(* Logix 5000 project; controller Safety vendor 1 type 14 code 86 rev 19.11; software revision 19.01; part 2 of 17 *)
(* tags used below, declared in another part *)
   A1_IO : UDT_CardSts[32];   // A1 Point I/O
   A1_IOSts_Flt : BOOL;   // A1 Point IO Module Fault ( 1= Faulted)
   C1_IO : UDT_CardSts[32];   // C1 Point I/O
   C1_IOSts_Flt : BOOL;   // C1 Point IO Module Fault ( 1= Faulted)
   CHPLC_IO : UDT_CardSts[32];   // CHPLC Point I/O
   CHPLC_IOSts_Flt : BOOL;   // CHPLC Point IO Module Fault ( 1= Faulted)
   D1_IO : UDT_CardSts[32];   // D1 Point I/O
   D1_IOSts_Flt : BOOL;   // D1 Point IO Module Fault ( 1= Faulted)
   DPD_IO : UDT_CardSts[32];   // DPD Point I/O
   DPD_IOSts_Flt : BOOL;   // DPD Point IO Module Fault ( 1= Faulted)
   E1_IO : UDT_CardSts[32];   // E1 Point I/O
   E1_IOSts_Flt : BOOL;   // E1 Point IO Module Fault ( 1= Faulted)
   F1_IO : UDT_CardSts[32];   // F1 Point I/O
   F1_IOSts_Flt : BOOL;   // F1 Point IO Module Fault ( 1= Faulted)
   Flt_Modules : DINT[5];   // Point IO Module Fault Word
   G1_IO : UDT_CardSts[32];   // G1 Point I/O
   G1_IOSts_Flt : BOOL;   // G1 Point IO Module Fault ( 1= Faulted)
   H1_IO : UDT_CardSts[32];   // H1 Point I/O
   H1_IOSts_Flt : BOOL;   // H1 Point IO Module Fault ( 1= Faulted)
   Line_TotalMode : BOOL;   // Line TOTAL Mode ( 1= Total Mode) (0 = Coil to Coil)
   LineSts : UDT_SysStatus;
   Local_ModFlts : DINT;   // Local Card Fault Status
   Local_Networks_OK : BOOL;   // Local Network CARDS OK ( 1= OK)
   Local_Slot : UDT_CardSts[17];   // Safety Processor
   MCC1_IO : UDT_CardSts[32];   // MCC1 Point I/O
   MCC1_IOSts_Flt : BOOL;   // MCC1 Point IO Module Fault ( 1= Faulted)
   MCC3_IO : UDT_CardSts[32];   // MCC3 Point I/O
   MCC4_IO : UDT_CardSts[32];   // MCC4 Point I/O
   OS11_IO : UDT_CardSts[32];   // OS11 Point I/O
   OS13_IO : UDT_CardSts[32];   // OS13 Point I/O
   OS14_IO : UDT_CardSts[32];   // OS14 Point I/O
   OS15_IO : UDT_CardSts[32];   // OS15 Point I/O
   OS16_IO : UDT_CardSts[32];   // OS16 Point I/O
   OS1_IO : UDT_CardSts[32];   // OS1 Point I/O
   OS2_IO : UDT_CardSts[32];   // OS2 Point I/O
   OS3_IO : UDT_CardSts[32];   // OS3 Point I/O
   OS4N_IO : UDT_CardSts[32];   // OS4N Point I/O
   OS4S_IO : UDT_CardSts[32];   // OS4S Point I/O
   OS5_IO : UDT_CardSts[32];   // OS5 Point I/O
   OS6_IO : UDT_CardSts[32];   // OS6 Point I/O
   OS8_IO : UDT_CardSts[32];   // OS8 Point I/O
   OS9_IO : UDT_CardSts[32];   // OS9 Point I/O
   Peer_Networks_OK : BOOL;   // Peer Network CARDS OK ( 1= OK)
   Rem_ModFlts : DINT;   // Remote IO Comm Faults
   SDPLC_IO : UDT_CardSts[32];   // SDPLC Point I/O
   SftyMap_Mach : DINT[5];   // SAFETY MAPPED From Machine Processor
   Sy_ClrFlt : BOOL;   // System Clear Fault

   UNW_SafeOffFltRst : BOOL;   // Unwind Safe-Off Fault Reset ( 1= Reset Cmd )
   UnwHoldDwn_FVR_En : BOOL := 1;   // Unwind Hold Down Roll FVR Enable ( 1= Enable )
   UnwHoldDwn_FVR_FltRst : BOOL;   // Unwind Hold Down Roll Fault Reset ( 1= Reset Cmd )
   UnwHoldDwn_FVR_FwdCmd : BOOL;   // Unwind Hold Down Roll Forward Command ( 1= Run Fwd )
   UnwHoldDwn_FVR_RevCmd : BOOL;   // Unwind Hold Down Roll Reverse Command ( 1= Run Rev)
   UWCC_Rst_PB : ALIAS FOR SftyMap_Mach[0].10;   // Unwind Coil Car Safety Reset PB
   VS2_IO : UDT_CardSts[32] := ([0].EntrySts := 16897, [0].Running := 1);   // VS2 Point I/O
        [4]   // 1734-IE2C/C
   VS2_IOSts_Flt : BOOL;   // VS2 Point IO Module Fault ( 1= Faulted)
   VS2_S10_ModFlt : ALIAS FOR Flt_Modules[0].21;   // VS2 Point I/O Slot10 Module Fault (1 = Fault)
   VS2_SolPwrEn : BOOL := 1;   // VS2 Solenoid Safe-Off Enable ( 1= Enable )
   WTPR_DrvsOff : BOOL;   // Wash Tank Pinch Rolls (1-4) Drives OFF ( 1= OFF)
   WTPR_SafeTrqEn : BOOL := 1;   // Wash Tank Pinch Rolls (1-4) Safe-Trq Off Enable ( 1= Enable )
   x172CR460 : ALIAS FOR SDPLC:1:I.Pt00Data;   // Shear Die Drive Main Contactor Safety Relay Input
   x172CR510 : ALIAS FOR SDPLC:1:I.Pt01Data;   // Shear Die Drive Enable Safety Relay Input
   x201PB040a : ALIAS FOR OS1:1:I.Pt00Data;   // Line Emergency Stop PB
   x201PB040b : ALIAS FOR OS1:1:I.Pt01Data;   // Line Emergency Stop PB
   x211PB040a : ALIAS FOR OS2:1:I.Pt00Data;   // Line Emergency Stop PB
   x211PB040b : ALIAS FOR OS2:1:I.Pt01Data;   // Line Emergency Stop PB
   x221PB040a : ALIAS FOR OS3:1:I.Pt00Data;   // Emergency Stop PB
   x221PB040b : ALIAS FOR OS3:1:I.Pt01Data;   // Emergency Stop PB
   x231PB040a : ALIAS FOR OS4N:1:I.Pt00Data;   // Emergency Stop PB
   x231PB040b : ALIAS FOR OS4N:1:I.Pt01Data;   // Emergency Stop PB
   x241PB040a : ALIAS FOR OS4S:1:I.Pt00Data;   // Emergency Stop PBMc_A_Run1_A
   x241PB040b : ALIAS FOR OS4S:1:I.Pt01Data;   // Emergency Stop PBMc_A_Run1_A
   x251PB040a : ALIAS FOR OS5:1:I.Pt00Data;   // Emergency Stop PB
   x251PB040b : ALIAS FOR OS5:1:I.Pt01Data;   // Emergency Stop PB
   x261PB040a : ALIAS FOR OS6:1:I.Pt00Data;   // Emergency Stop PB
   x261PB040b : ALIAS FOR OS6:1:I.Pt01Data;   // Emergency Stop PB
   x271PB040a : ALIAS FOR OS8:1:I.Pt00Data;   // Emergency Stop PB
   x271PB040b : ALIAS FOR OS8:1:I.Pt01Data;   // Emergency Stop PB
   x281PB040a : ALIAS FOR OS9:1:I.Pt00Data;   // Emergency Stop PB
   x281PB040b : ALIAS FOR OS9:1:I.Pt01Data;   // Emergency Stop PB
   x291PB040a : ALIAS FOR OS11:1:I.Pt00Data;   // Emergency Stop PB
   x291PB040b : ALIAS FOR OS11:1:I.Pt01Data;   // Emergency Stop PB
   x301PB040a : ALIAS FOR OS13:1:I.Pt00Data;   // Emergency Stop PB
   x301PB040b : ALIAS FOR OS13:1:I.Pt01Data;   // Emergency Stop PB
   x301PBL500 : BOOL;   // Tandem Jog PBL
   x301SS540a : BOOL;   // Sheeter Pinch Roll Jog Forward SS
   x301SS540b : BOOL;   // Sheeter Pinch Roll Jog Reverse SS
   x311PB040a : ALIAS FOR OS14:1:I.Pt00Data;   // Emergency Stop PB OS14
   x311PB040b : ALIAS FOR OS14:1:I.Pt01Data;   // Emergency Stop PB OS14
   x311PB130a : ALIAS FOR OS14:1:I.Pt02Data;   // Shear Emergency Stop PB Os14
   x311PB130b : ALIAS FOR OS14:1:I.Pt03Data;   // Shear Emergency Stop PB Os14
   x312PB700 : BOOL;   // Product Conveyor Jog Forward PB
   x312PB740 : BOOL;   // Product Conveyor Jog Reverse PB
   x312SS460a : BOOL;   // Scrap Conveyor Jog Forward SS
   x312SS460b : BOOL;   // Scrap Conveyor Jog Reverse SS
   x313PBL080 : BOOL;   // Tandem Jog PBL
   x313SS460a : BOOL;   // Shear Conveyor Jog Forward SS
   x313SS460b : BOOL;   // Shear Conveyor Jog Reverse SS
   x314SS040a : BOOL;   // Shear Pinch Roll Jog Forward SS
   x314SS040b : BOOL;   // Shear Pinch Roll Jog Reverse SS
   x315SS040a : BOOL;   // Sheeter Pinch Roll Jog Forward SS
   x315SS040b : BOOL;   // Sheeter Pinch Roll Jog Reverse SS
   x321PB040a : ALIAS FOR OS15:1:I.Pt00Data;   // Emergency Stop PB
   x321PB040b : ALIAS FOR OS15:1:I.Pt01Data;   // Emergency Stop PB
   x331PB040a : ALIAS FOR OS16:1:I.Pt00Data;   // Emergency Stop PB
   x331PB040b : ALIAS FOR OS16:1:I.Pt01Data;   // Emergency Stop PB
   x406LCA047 : ALIAS FOR A1:21:I.Pt00Data;   // North/South Light Curtain Output A
   x406LCB052 : ALIAS FOR A1:21:I.Pt01Data;   // North/South Light Curtain Output B
   x480PB470a : ALIAS FOR DPD:15:I.Pt00Data;   // Emergency Stop Pushbutton
   x480PB470b : ALIAS FOR DPD:15:I.Pt01Data;   // Emergency Stop Pushbutton
   x480PB550a : ALIAS FOR DPD:15:I.Pt02Data;   // Emergency Stop Pushbutton (In Pit)
   x480PB550b : ALIAS FOR DPD:15:I.Pt03Data;   // Emergency Stop Pushbutton (In Pit)
   x519LS470 : ALIAS FOR G1:12:I.Pt00Data;   // Tripwire Emergency Stop Limit Switch
   x533PB470a : ALIAS FOR H1:6:I.Pt00Data;   // Sheeter Emergency Stop Pushbutton
   x533PB470b : ALIAS FOR H1:6:I.Pt01Data;   // Sheeter Emergency Stop Pushbutton
   x613CR460 : ALIAS FOR CHPLC:1:I.Pt00Data;   // Unwind Operator Side Main Contactor Safety Relay
   x613CR510 : ALIAS FOR CHPLC:1:I.Pt01Data;   // Unwind Operator Side Drive Enable Safety Relay
   x613CR550 : ALIAS FOR CHPLC:1:I.Pt02Data;   // Unwind Drive Side Main Contactor Safety Relay
   x613CR590 : ALIAS FOR CHPLC:1:I.Pt03Data;   // Unwind Drive Side Drive Enable Safety Relay
   x613CR630 : ALIAS FOR CHPLC:1:I.Pt04Data;   // #1 Entry Bridle Roll 2 Main Contactor Safety Relay
   x613CR670 : ALIAS FOR CHPLC:1:I.Pt05Data;   // #1 Entry Bridle Roll 2 Drive Enable Safety Relay
   x613CR710 : ALIAS FOR CHPLC:1:I.Pt06Data;   // #2 Entry Bridle Roll 3 Main Contactor Safety Relay
   x613CR750 : ALIAS FOR CHPLC:1:I.Pt07Data;   // #2 Entry Bridle Roll 3 Drive Enable Safety Relay
   x614CR040 : ALIAS FOR CHPLC:2:I.Pt00Data;   // #1 Exit Bridle Roll 6 Main Contactor Safety Relay
   x614CR090 : ALIAS FOR CHPLC:2:I.Pt01Data;   // #1 Exit Bridle Roll 6 Drive Enable Safety Relay
   x614CR130 : ALIAS FOR CHPLC:2:I.Pt02Data;   // #2 Exit Bridle Roll 7 Main Contactor Safety Relay
   x614CR170 : ALIAS FOR CHPLC:2:I.Pt03Data;   // #2 Exit Bridle Roll 7 Drive Enable Safety Relay
   x614CR210 : ALIAS FOR CHPLC:2:I.Pt04Data;   // Rewind Main Contactor Safety Relay
   x614CR250 : ALIAS FOR CHPLC:2:I.Pt05Data;   // Rewind Drive Enable Safety Relay
   x702MTR191FF : ALIAS FOR MCC1:1:I.Pt00Data;   // Rewind Pinch Roll Fwd Fdbk
   x702MTR191RF : ALIAS FOR MCC1:1:I.Pt01Data;   // Rewind Pinch Roll Rev Fdbk
   x708MTR080FF : ALIAS FOR MCC1:1:I.Pt04Data;   // Flattener Drive Motor Fwd Fdbk
   x708MTR080RF : ALIAS FOR MCC1:1:I.Pt05Data;   // Flattener Drive Motor Rev Fdbk
   x708MTR250FF : ALIAS FOR MCC1:1:I.Pt06Data;   // Unwind Holddown Roll Drive Motor Fwd Fdbk
   x708MTR250RF : ALIAS FOR MCC1:1:I.Pt07Data;   // Unwind Holddown Roll Drive Motor Rev Fdbk
   x753MTR190FF : ALIAS FOR MCC3:1:I.Pt00Data;   // Trimmer Pinch Roll Fwd Fdbk
   x753MTR190RF : ALIAS FOR MCC3:1:I.Pt01Data;   // Trimmer Pinch Roll Rev Fdbk
   x759MTR080SE : ALIAS FOR MCC3:4:O.Pt02Data;   // Scrap Choppers Width Adjust Safety Enable
   x759MTR080SP : ALIAS FOR MCC3:4:O.Pt01Data;   // Scrap Choppers Width Adjust Safety Power
   x761MTR081RF : ALIAS FOR MCC3:1:I.Pt02Data;   // Trimmer Scrap Conveyor RunFdbk
   x775MTR280RF : BOOL := 1;   // (From Shear DIe) Shear Pinch Roll Lube Run Fdbk
   x778MTR080RF : ALIAS FOR MCC4:1:I.Pt00Data;   // Shear Crank Motor Run Fdbk
   x781MTR080RF : BOOL := 1;   // (From Shear DIe) Sheeter Pinch Roll Lube Run Fdbk
   x781MTR190RF : BOOL := 1;   // (From Shear DIe) Sheeter Hyd Pump Run Fdbk
   x802MTR080FF : ALIAS FOR MCC5:1:I.Pt00Data;   // Stacker Side Guide Lift Fwd Fdbk/Up
   x802MTR080RF : ALIAS FOR MCC5:1:I.Pt01Data;   // Stacker Side Guide Lift Rev Fdbk/Down
   x802MTR230FF : ALIAS FOR MCC5:1:I.Pt02Data;   // Scrap Horizontal Conveyor Run Fwd Fdbk
   x802MTR230RF : ALIAS FOR MCC5:1:I.Pt03Data;   // Scrap Horizontal Conveyor Run Rev Fdbk
   x802MTR231FF : ALIAS FOR MCC5:1:I.Pt04Data;   // Stacker Chain Fwd Fdbk
   x802MTR231RF : ALIAS FOR MCC5:1:I.Pt05Data;   // Stacker Chain Rev Fdbk
   x813MTR080RF : BOOL := 1;   // (From Shear DIe) Exit Conveyor Hyd Pump Run Fdbk
   y172CR460 : ALIAS FOR SDPLC:2:O.Pt00Data;   // Shear Die Drive Main Contactor Safety Relay Output
   y172CR510 : ALIAS FOR SDPLC:2:O.Pt01Data;   // Shear Die Drive Enable Safety Relay Output
   y172CR550 : ALIAS FOR SDPLC:2:O.Pt02Data;   // Line Soleniod Safe-Off
   y233CR040 : ALIAS FOR OS4N:5:O.Pt00Data;   // OS4N Solenoid Safe Off
   y243CR040 : ALIAS FOR OS4S:5:O.Pt00Data;   // OS4S Solenoid Safe Off
   y406CR050 : ALIAS FOR A1:20:O.Pt00Data;   // Line Solenoid Safe Off
   y406CR090 : ALIAS FOR A1:20:O.Pt01Data;   // Coil Car Solenoid Safe Off
   y406CR120 : ALIAS FOR A1:20:O.Pt02Data;   // Spare
   y406CR170 : ALIAS FOR A1:20:O.Pt03Data;   // Spare
   y435CR050 : ALIAS FOR C1:12:O.Pt00Data;   // Solenoid Safe Off
   y451CR050 : ALIAS FOR D1:12:O.Pt00Data;   // Soleniod Safe Off
   y464CR050 : ALIAS FOR E1:10:O.Pt00Data;   // Soleniod Safe Off
   y480CR050 : ALIAS FOR DPD:14:O.Pt00Data;   // Solenoid Safe Off
   y495CR050 : ALIAS FOR VS2:10:O.Pt00Data;   // Soleniod Safe Off
   y507CR050 : ALIAS FOR F1:19:O.Pt00Data;   // Line Solenoid Safe Off
   y507CR090 : ALIAS FOR F1:19:O.Pt01Data;   // Rewind Coil Car Solenoid Safe Off
   y519CR050 : ALIAS FOR G1:11:O.Pt00Data;   // Line Solenoid Safe Off
   y533CR050 : ALIAS FOR H1:5:O.Pt00Data;   // Line Solenoid Safe Off
   y613CR460 : ALIAS FOR CHPLC:4:O.Pt00Data;   // Unwind Operator Side Main Contactor Safety Relay
   y613CR510 : ALIAS FOR CHPLC:4:O.Pt01Data;   // Unwind Operator Side Drive Enable Safety Relay
   y613CR550 : ALIAS FOR CHPLC:4:O.Pt02Data;   // Unwind Drive Side Main Contactor Safety Relay
   y613CR590 : ALIAS FOR CHPLC:4:O.Pt03Data;   // Unwind Drive Side Drive Enable Safety Relay
   y613CR630 : ALIAS FOR CHPLC:4:O.Pt04Data;   // #1 Entry Bridle Roll 2 Main Contactor Safety Relay
   y613CR670 : ALIAS FOR CHPLC:4:O.Pt05Data;   // #1 Entry Bridle Roll 2 Drive Enable Safety Relay
   y613CR710 : ALIAS FOR CHPLC:4:O.Pt06Data;   // #2 Entry Bridle Roll 3 Main Contactor Safety Relay
   y613CR750 : ALIAS FOR CHPLC:4:O.Pt07Data;   // #2 Entry Bridle Roll 3 Drive Enable Safety Relay
   y614CR040 : ALIAS FOR CHPLC:5:O.Pt00Data;   // #1 Exit Bridle Roll 6 Main Contactor Safety Relay
   y614CR090 : ALIAS FOR CHPLC:5:O.Pt01Data;   // #1 Exit Bridle Roll 6 Drive Enable Safety Relay
   y614CR130 : ALIAS FOR CHPLC:5:O.Pt02Data;   // #2 Exit Bridle Roll 7 Main Contactor Safety Relay
   y614CR170 : ALIAS FOR CHPLC:5:O.Pt03Data;   // #2 Exit Bridle Roll 7 Drive Enable Safety Relay
   y614CR210 : ALIAS FOR CHPLC:5:O.Pt04Data;   // Rewind Main Contactor Safety Relay
   y614CR250 : ALIAS FOR CHPLC:5:O.Pt05Data;   // Rewind Drive Enable Safety Relay
   y702MTR191FC : ALIAS FOR MCC1:6:O.Pt00Data;   // Rewind Pinch Roll Fwd Cmd
   y702MTR191RC : ALIAS FOR MCC1:6:O.Pt01Data;   // Rewind Pinch Roll Rev Cmd
   y708MTR080FC : ALIAS FOR MCC1:6:O.Pt04Data;   // Flattener Drive Motor Fwd Cmd
   y708MTR080RC : ALIAS FOR MCC1:6:O.Pt05Data;   // Flattener Drive Motor Rev Cmd
   y708MTR250FC : ALIAS FOR MCC1:6:O.Pt06Data;   // Unwind Holddown Roll Drive Motor Fwd Cmd
   y708MTR250RC : ALIAS FOR MCC1:6:O.Pt07Data;   // Unwind Holddown Roll Drive Motor Rev Cmd
   y725MTR080SE : ALIAS FOR MCC2:1:O.Pt01Data;   // Unwind Pinch Roll Safety Enable
   y725MTR080SP : ALIAS FOR MCC2:1:O.Pt00Data;   // Unwind Pinch Roll Safety Power
   y727MTR080SE : ALIAS FOR MCC2:1:O.Pt05Data;   // Paper Winder Safety Enable
   y727MTR080SP : ALIAS FOR MCC2:1:O.Pt04Data;   // Paper Winder Safety Power
   y729MTR080SE : ALIAS FOR MCC2:1:O.Pt03Data;   // Washtank Pinch Roll 4 Safety Enable
   y729MTR080SP : ALIAS FOR MCC2:1:O.Pt02Data;   // Washtank Pinch Roll 4 Safety Power
   y731MTR080SE : ALIAS FOR MCC2:1:O.Pt07Data;   // Washtank Pinch Roll 1 Safety Enable
   y731MTR080SP : ALIAS FOR MCC2:1:O.Pt06Data;   // Washtank Pinch Roll 1 Safety Power
   y733MTR080SE : ALIAS FOR MCC2:2:O.Pt01Data;   // Washtank Pinch Roll 2 Safety Enable
   y733MTR080SP : ALIAS FOR MCC2:2:O.Pt00Data;   // Washtank Pinch Roll 2 Safety Power
   y735MTR080SE : ALIAS FOR MCC2:2:O.Pt03Data;   // Washtank Pinch Roll 3 Safety Enable
   y735MTR080SP : ALIAS FOR MCC2:2:O.Pt02Data;   // Washtank Pinch Roll 3 Safety Power
   y751MTR080SE : ALIAS FOR MCC3:3:O.Pt04Data;   // Trimmer Knives Safety Enable
   y751MTR080SP : ALIAS FOR MCC3:3:O.Pt03Data;   // Trimmer Knives Safety Power
   y753MTR190FC : ALIAS FOR MCC3:3:O.Pt00Data;   // Trimmer Pinch Roll Fwd Cmd
   y753MTR190RC : ALIAS FOR MCC3:3:O.Pt01Data;   // Trimmer Pinch Roll Rev Cmd
   y754MTR080SE : ALIAS FOR MCC3:3:O.Pt06Data;   // Side Guide Width Adjust Safety Enable
   y754MTR080SP : ALIAS FOR MCC3:3:O.Pt05Data;   // Side Guide Width Adjust Safety Power
   y755MTR080SE : ALIAS FOR MCC3:4:O.Pt00Data;   // Trimmer Knives Width Adjust Safety Enable
   y755MTR080SP : ALIAS FOR MCC3:3:O.Pt07Data;   // Trimmer Knives Width Adjust Safety Power
   y761MTR081RC : ALIAS FOR MCC3:3:O.Pt02Data;   // Trimmer Scrap Conveyor RunCmd
   y762MTR080SE : ALIAS FOR MCC3:4:O.Pt04Data;   // Scrap Choppers Safety Enable
   y762MTR080SP : ALIAS FOR MCC3:4:O.Pt03Data;   // Scrap Choppers Safety Power
   y776MTR080SE : ALIAS FOR MCC4:3:O.Pt07Data;   // Shear Metering Backup Roll Safety Enable
   y776MTR080SP : ALIAS FOR MCC4:3:O.Pt06Data;   // Shear Metering Backup Roll Safety Power
   y778MTR080RC : ALIAS FOR MCC4:4:O.Pt00Data;   // Shear Die Crank Run Cmd
   y779MTR080SE : ALIAS FOR MCC4:3:O.Pt01Data;   // Shear Pinch Roll Safety Enable
   y779MTR080SP : ALIAS FOR MCC4:3:O.Pt00Data;   // Shear Pinch Roll Safety Power
   y782MTR080SE : ALIAS FOR MCC4:3:O.Pt03Data;   // Sheeter Pinch Roll Safety Enable
   y782MTR080SP : ALIAS FOR MCC4:3:O.Pt02Data;   // Sheeter Pinch Roll Safety Power
   y785MTR080SE : ALIAS FOR MCC4:3:O.Pt05Data;   // Stacker Blower Safety Enable
   y785MTR080SP : ALIAS FOR MCC4:3:O.Pt04Data;   // Stacker Blower Safety Power
   y800MTR080SE : ALIAS FOR MCC5:3:O.Pt01Data;   // Scrap Incline Conveyor Safety Enable
   y800MTR080SP : ALIAS FOR MCC5:3:O.Pt00Data;   // Scrap Incline Conveyor Safety Power
   y802MTR080FC : ALIAS FOR MCC5:4:O.Pt04Data;   // Stacker Side Guide Lift Fwd Cmd/Up
   y802MTR080RC : ALIAS FOR MCC5:4:O.Pt05Data;   // Stacker Side Guide Lift Rev Cmd/Down
   y802MTR230FC : ALIAS FOR MCC5:4:O.Pt06Data;   // Scrap Horizontal Conveyor Fwd Cmd
   y802MTR230RC : ALIAS FOR MCC5:4:O.Pt07Data;   // Scrap Horizontal Conveyor Rev Cmd
   y802MTR231FC : ALIAS FOR MCC5:5:O.Pt00Data;   // Stacker Chain Fwd Cmd
   y802MTR231RC : ALIAS FOR MCC5:5:O.Pt01Data;   // Stacker Chain Rev Cmd
   y804MTR080SE : ALIAS FOR MCC5:3:O.Pt03Data;   // Stacker Back Stop Safety Enable
   y804MTR080SP : ALIAS FOR MCC5:3:O.Pt02Data;   // Stacker Back Stop Safety Power
   y806MTR080SE : ALIAS FOR MCC5:3:O.Pt05Data;   // Product Conveyor 3 Safety Enable
   y806MTR080SP : ALIAS FOR MCC5:3:O.Pt04Data;   // Product Conveyor 3 Safety Power
   y808MTR080SE : ALIAS FOR MCC5:3:O.Pt07Data;   // Product Conveyor 1 Safety Enable
   y808MTR080SP : ALIAS FOR MCC5:3:O.Pt06Data;   // Product Conveyor 1 Safety Power
   y810MTR080SE : ALIAS FOR MCC5:4:O.Pt01Data;   // Product Conveyor 2 Safety Enable
   y810MTR080SP : ALIAS FOR MCC5:4:O.Pt00Data;   // Product Conveyor 2 Safety Power
   y812MTR080SE : ALIAS FOR MCC5:4:O.Pt03Data;   // Shear Conveyor Safety Enable
   y812MTR080SP : ALIAS FOR MCC5:4:O.Pt02Data;   // Shear Conveyor Safety Power
END_VAR

PROGRAM CardSts   (* main routine Main *)
// Local and Remote IO
// Card Status

ROUTINE A1_IO   (* ladder *)
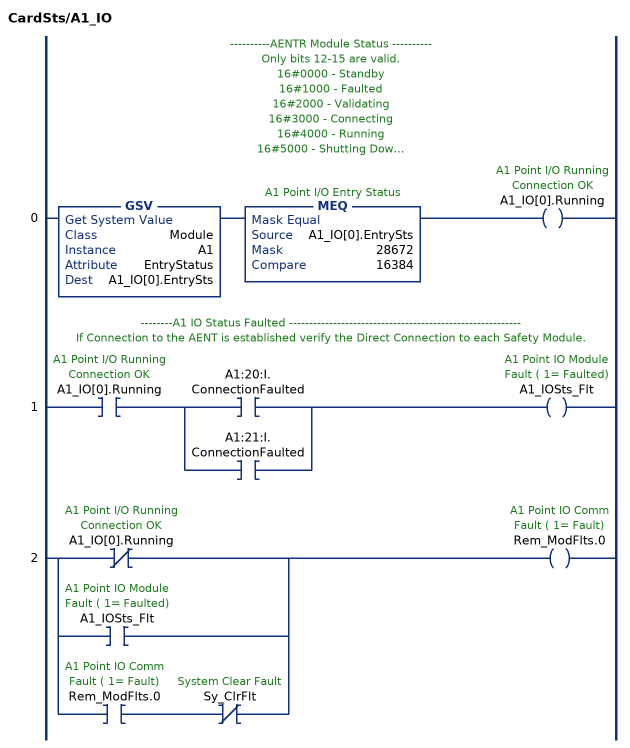
   // ----------AENTR Module Status ----------
   // Only bits 12-15 are valid.
   // 16#0000 - Standby
   // 16#1000 - Faulted
   // 16#2000 - Validating
   // 16#3000 - Connecting
   // 16#4000 - Running
   // 16#5000 - Shutting Down
   // 16#6000 - Inhibited
   // 16#7000 - Waiting
   0: GSV(Module,A1,EntryStatus,A1_IO[0].EntrySts)MEQ(A1_IO[0].EntrySts,28672,16384)OTE(A1_IO[0].Running);
   // --------A1 IO Status Faulted ----------------------------------------------------------
   // If Connection to the AENT is established verify the Direct Connection to each Safety Module.
   1: XIC(A1_IO[0].Running)[XIC(A1:20:I.ConnectionFaulted) ,XIC(A1:21:I.ConnectionFaulted) ]OTE(A1_IOSts_Flt);
   2: [XIO(A1_IO[0].Running) ,XIC(A1_IOSts_Flt) ,XIC(Rem_ModFlts.0) XIO(Sy_ClrFlt) ]OTE(Rem_ModFlts.0);
END_ROUTINE

ROUTINE C1_IO   (* ladder *)
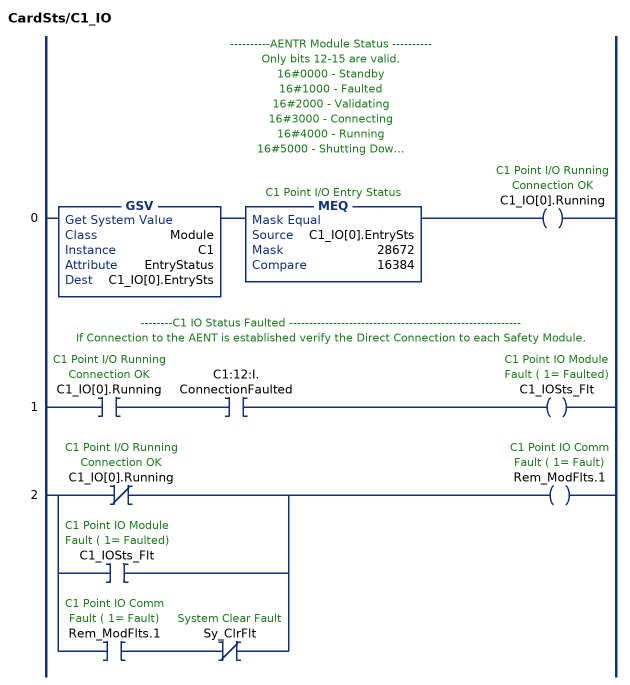
   // ----------AENTR Module Status ----------
   // Only bits 12-15 are valid.
   // 16#0000 - Standby
   // 16#1000 - Faulted
   // 16#2000 - Validating
   // 16#3000 - Connecting
   // 16#4000 - Running
   // 16#5000 - Shutting Down
   // 16#6000 - Inhibited
   // 16#7000 - Waiting
   0: GSV(Module,C1,EntryStatus,C1_IO[0].EntrySts)MEQ(C1_IO[0].EntrySts,28672,16384)OTE(C1_IO[0].Running);
   // --------C1 IO Status Faulted ----------------------------------------------------------
   // If Connection to the AENT is established verify the Direct Connection to each Safety Module.
   1: XIC(C1_IO[0].Running)XIC(C1:12:I.ConnectionFaulted)OTE(C1_IOSts_Flt);
   2: [XIO(C1_IO[0].Running) ,XIC(C1_IOSts_Flt) ,XIC(Rem_ModFlts.1) XIO(Sy_ClrFlt) ]OTE(Rem_ModFlts.1);
END_ROUTINE

ROUTINE CHPLC_IO   (* ladder *)
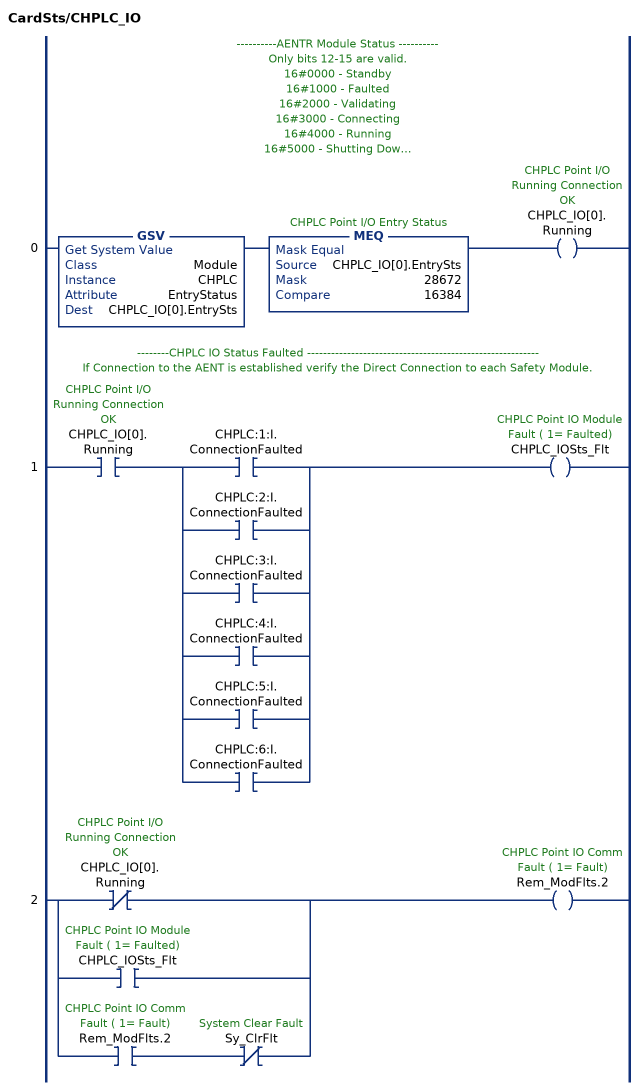
   // ----------AENTR Module Status ----------
   // Only bits 12-15 are valid.
   // 16#0000 - Standby
   // 16#1000 - Faulted
   // 16#2000 - Validating
   // 16#3000 - Connecting
   // 16#4000 - Running
   // 16#5000 - Shutting Down
   // 16#6000 - Inhibited
   // 16#7000 - Waiting
   0: GSV(Module,CHPLC,EntryStatus,CHPLC_IO[0].EntrySts)MEQ(CHPLC_IO[0].EntrySts,28672,16384)OTE(CHPLC_IO[0].Running);
   // --------CHPLC IO Status Faulted ----------------------------------------------------------
   // If Connection to the AENT is established verify the Direct Connection to each Safety Module.
   1: XIC(CHPLC_IO[0].Running)[XIC(CHPLC:1:I.ConnectionFaulted) ,XIC(CHPLC:2:I.ConnectionFaulted) ,XIC(CHPLC:3:I.ConnectionFaulted) ,XIC(CHPLC:4:I.ConnectionFaulted) ,XIC(CHPLC:5:I.ConnectionFaulted) ,XIC(CHPLC:6:I.ConnectionFaulted) ]OTE(CHPLC_IOSts_Flt);
   2: [XIO(CHPLC_IO[0].Running) ,XIC(CHPLC_IOSts_Flt) ,XIC(Rem_ModFlts.2) XIO(Sy_ClrFlt) ]OTE(Rem_ModFlts.2);
END_ROUTINE

ROUTINE D1_IO   (* ladder *)
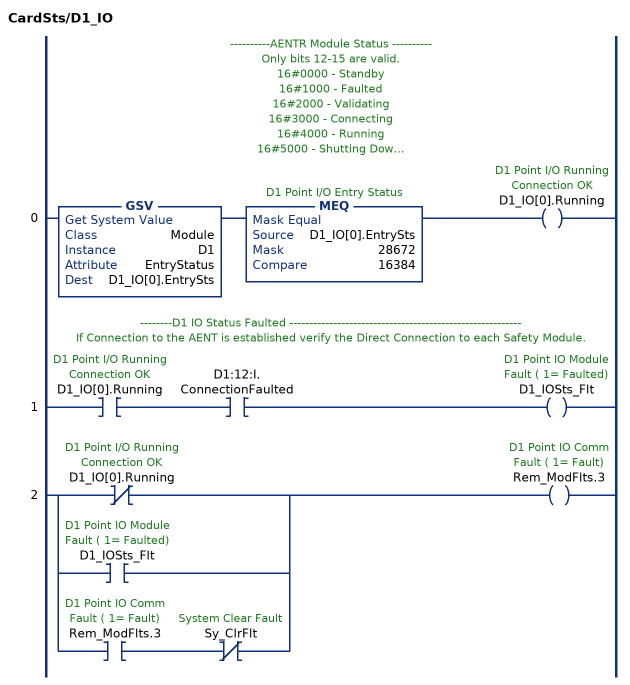
   // ----------AENTR Module Status ----------
   // Only bits 12-15 are valid.
   // 16#0000 - Standby
   // 16#1000 - Faulted
   // 16#2000 - Validating
   // 16#3000 - Connecting
   // 16#4000 - Running
   // 16#5000 - Shutting Down
   // 16#6000 - Inhibited
   // 16#7000 - Waiting
   0: GSV(Module,D1,EntryStatus,D1_IO[0].EntrySts)MEQ(D1_IO[0].EntrySts,28672,16384)OTE(D1_IO[0].Running);
   // --------D1 IO Status Faulted ----------------------------------------------------------
   // If Connection to the AENT is established verify the Direct Connection to each Safety Module.
   1: XIC(D1_IO[0].Running)XIC(D1:12:I.ConnectionFaulted)OTE(D1_IOSts_Flt);
   2: [XIO(D1_IO[0].Running) ,XIC(D1_IOSts_Flt) ,XIC(Rem_ModFlts.3) XIO(Sy_ClrFlt) ]OTE(Rem_ModFlts.3);
END_ROUTINE

ROUTINE DPD_IO   (* ladder *)
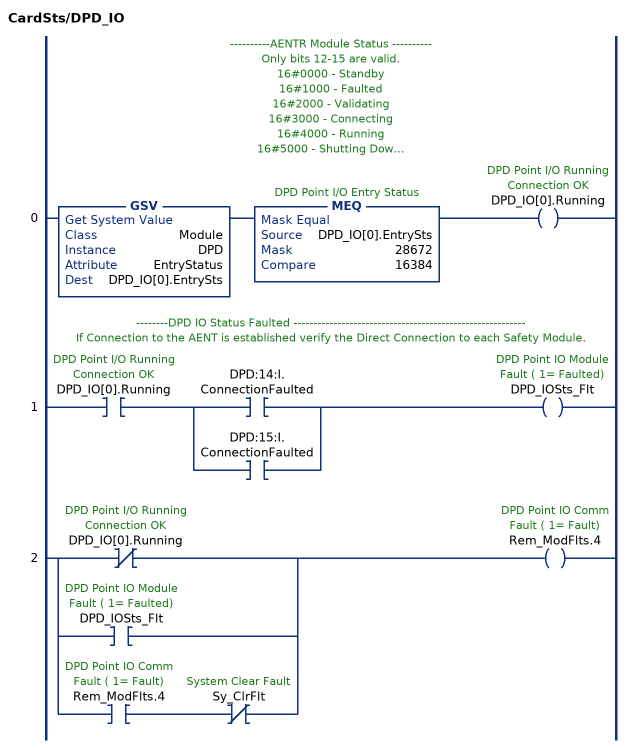
   // ----------AENTR Module Status ----------
   // Only bits 12-15 are valid.
   // 16#0000 - Standby
   // 16#1000 - Faulted
   // 16#2000 - Validating
   // 16#3000 - Connecting
   // 16#4000 - Running
   // 16#5000 - Shutting Down
   // 16#6000 - Inhibited
   // 16#7000 - Waiting
   0: GSV(Module,DPD,EntryStatus,DPD_IO[0].EntrySts)MEQ(DPD_IO[0].EntrySts,28672,16384)OTE(DPD_IO[0].Running);
   // --------DPD IO Status Faulted ----------------------------------------------------------
   // If Connection to the AENT is established verify the Direct Connection to each Safety Module.
   1: XIC(DPD_IO[0].Running)[XIC(DPD:14:I.ConnectionFaulted) ,XIC(DPD:15:I.ConnectionFaulted) ]OTE(DPD_IOSts_Flt);
   2: [XIO(DPD_IO[0].Running) ,XIC(DPD_IOSts_Flt) ,XIC(Rem_ModFlts.4) XIO(Sy_ClrFlt) ]OTE(Rem_ModFlts.4);
END_ROUTINE

ROUTINE E1_IO   (* ladder *)
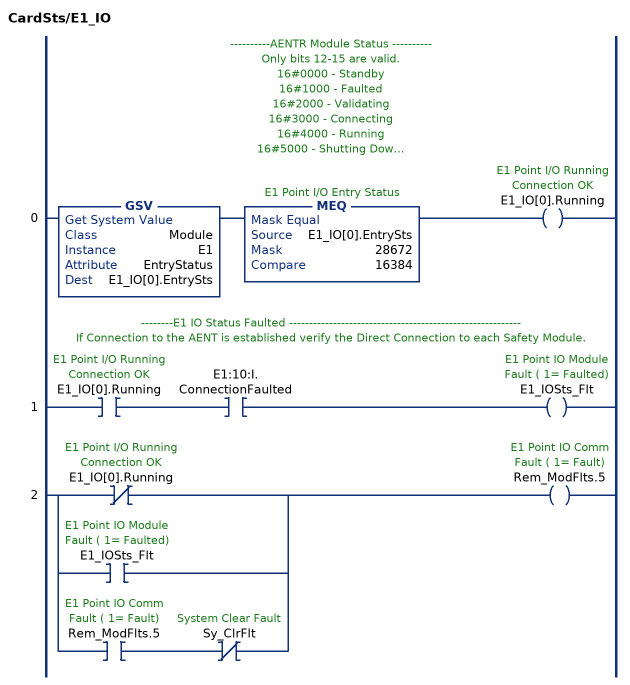
   // ----------AENTR Module Status ----------
   // Only bits 12-15 are valid.
   // 16#0000 - Standby
   // 16#1000 - Faulted
   // 16#2000 - Validating
   // 16#3000 - Connecting
   // 16#4000 - Running
   // 16#5000 - Shutting Down
   // 16#6000 - Inhibited
   // 16#7000 - Waiting
   0: GSV(Module,E1,EntryStatus,E1_IO[0].EntrySts)MEQ(E1_IO[0].EntrySts,28672,16384)OTE(E1_IO[0].Running);
   // --------E1 IO Status Faulted ----------------------------------------------------------
   // If Connection to the AENT is established verify the Direct Connection to each Safety Module.
   1: XIC(E1_IO[0].Running)XIC(E1:10:I.ConnectionFaulted)OTE(E1_IOSts_Flt);
   2: [XIO(E1_IO[0].Running) ,XIC(E1_IOSts_Flt) ,XIC(Rem_ModFlts.5) XIO(Sy_ClrFlt) ]OTE(Rem_ModFlts.5);
END_ROUTINE

ROUTINE F1_IO   (* ladder *)
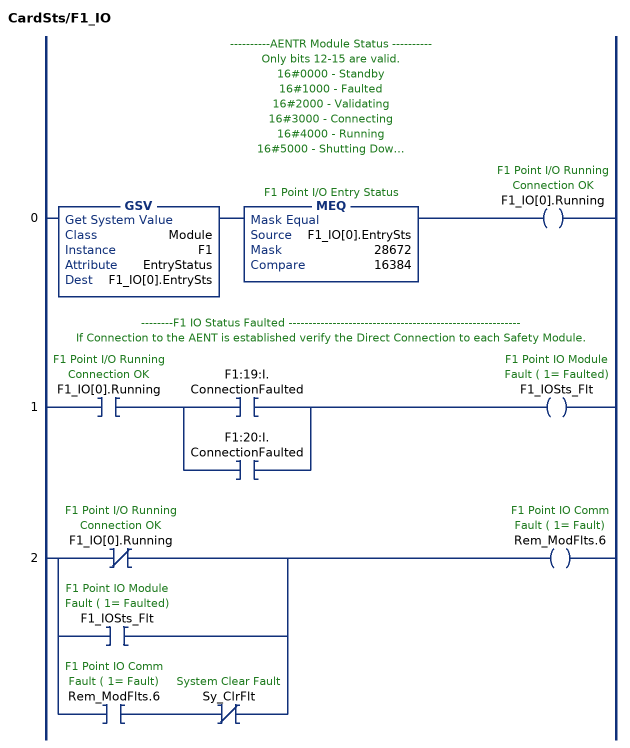
   // ----------AENTR Module Status ----------
   // Only bits 12-15 are valid.
   // 16#0000 - Standby
   // 16#1000 - Faulted
   // 16#2000 - Validating
   // 16#3000 - Connecting
   // 16#4000 - Running
   // 16#5000 - Shutting Down
   // 16#6000 - Inhibited
   // 16#7000 - Waiting
   0: GSV(Module,F1,EntryStatus,F1_IO[0].EntrySts)MEQ(F1_IO[0].EntrySts,28672,16384)OTE(F1_IO[0].Running);
   // --------F1 IO Status Faulted ----------------------------------------------------------
   // If Connection to the AENT is established verify the Direct Connection to each Safety Module.
   1: XIC(F1_IO[0].Running)[XIC(F1:19:I.ConnectionFaulted) ,XIC(F1:20:I.ConnectionFaulted) ]OTE(F1_IOSts_Flt);
   2: [XIO(F1_IO[0].Running) ,XIC(F1_IOSts_Flt) ,XIC(Rem_ModFlts.6) XIO(Sy_ClrFlt) ]OTE(Rem_ModFlts.6);
END_ROUTINE

ROUTINE G1_IO   (* ladder *)
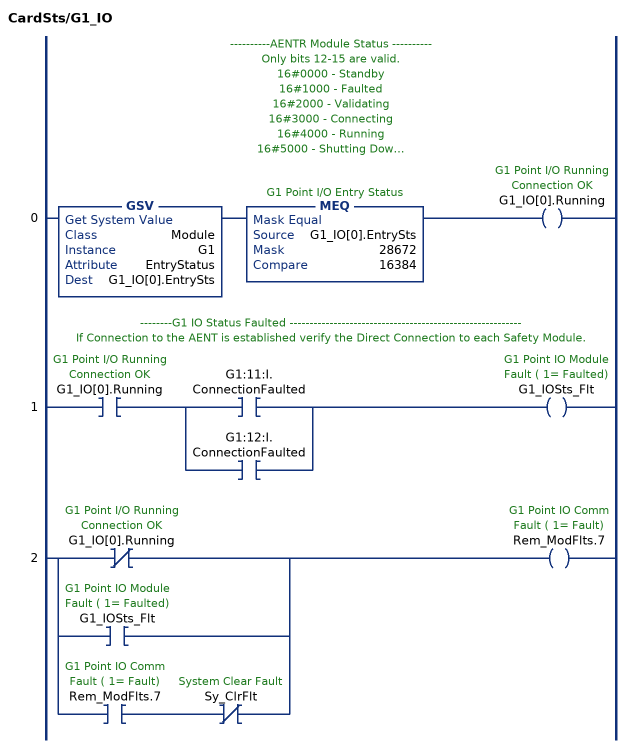
   // ----------AENTR Module Status ----------
   // Only bits 12-15 are valid.
   // 16#0000 - Standby
   // 16#1000 - Faulted
   // 16#2000 - Validating
   // 16#3000 - Connecting
   // 16#4000 - Running
   // 16#5000 - Shutting Down
   // 16#6000 - Inhibited
   // 16#7000 - Waiting
   0: GSV(Module,G1,EntryStatus,G1_IO[0].EntrySts)MEQ(G1_IO[0].EntrySts,28672,16384)OTE(G1_IO[0].Running);
   // --------G1 IO Status Faulted ----------------------------------------------------------
   // If Connection to the AENT is established verify the Direct Connection to each Safety Module.
   1: XIC(G1_IO[0].Running)[XIC(G1:11:I.ConnectionFaulted) ,XIC(G1:12:I.ConnectionFaulted) ]OTE(G1_IOSts_Flt);
   2: [XIO(G1_IO[0].Running) ,XIC(G1_IOSts_Flt) ,XIC(Rem_ModFlts.7) XIO(Sy_ClrFlt) ]OTE(Rem_ModFlts.7);
END_ROUTINE

ROUTINE H1_IO   (* ladder *)
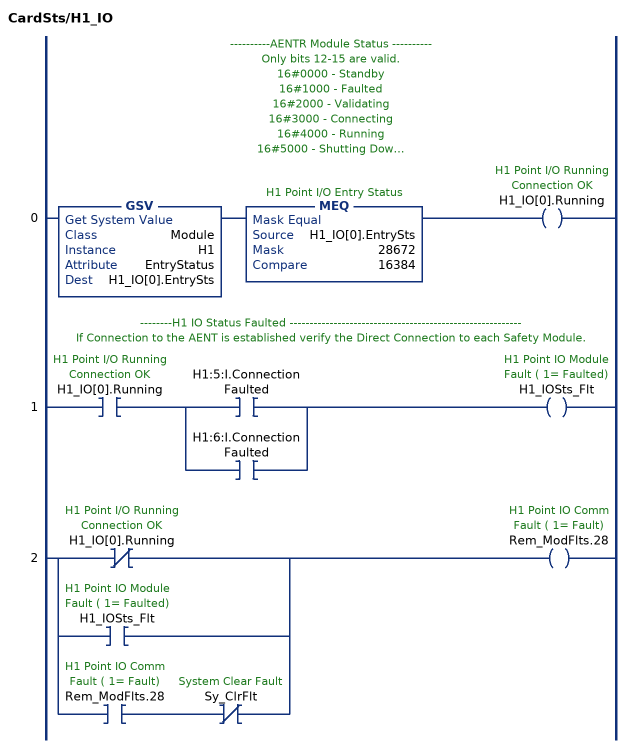
   // ----------AENTR Module Status ----------
   // Only bits 12-15 are valid.
   // 16#0000 - Standby
   // 16#1000 - Faulted
   // 16#2000 - Validating
   // 16#3000 - Connecting
   // 16#4000 - Running
   // 16#5000 - Shutting Down
   // 16#6000 - Inhibited
   // 16#7000 - Waiting
   0: GSV(Module,H1,EntryStatus,H1_IO[0].EntrySts)MEQ(H1_IO[0].EntrySts,28672,16384)OTE(H1_IO[0].Running);
   // --------H1 IO Status Faulted ----------------------------------------------------------
   // If Connection to the AENT is established verify the Direct Connection to each Safety Module.
   1: XIC(H1_IO[0].Running)[XIC(H1:5:I.ConnectionFaulted) ,XIC(H1:6:I.ConnectionFaulted) ]OTE(H1_IOSts_Flt);
   2: [XIO(H1_IO[0].Running) ,XIC(H1_IOSts_Flt) ,XIC(Rem_ModFlts.28) XIO(Sy_ClrFlt) ]OTE(Rem_ModFlts.28);
END_ROUTINE

ROUTINE Local_IO   (* ladder *)
// Local IO Card Status
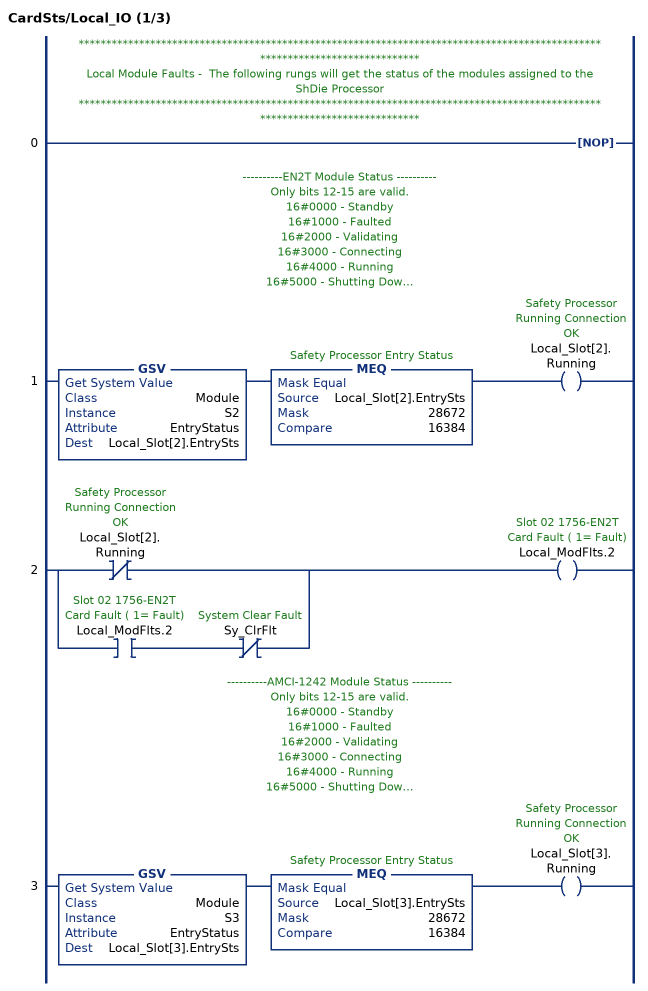
   // ****************************************************************************************************************************
   // Local Module Faults -  The following rungs will get the status of the modules assigned to the ShDie Processor
   // ****************************************************************************************************************************
   0: NOP();
   // ----------EN2T Module Status ----------
   // Only bits 12-15 are valid.
   // 16#0000 - Standby
   // 16#1000 - Faulted
   // 16#2000 - Validating
   // 16#3000 - Connecting
   // 16#4000 - Running
   // 16#5000 - Shutting Down
   // 16#6000 - Inhibited
   // 16#7000 - Waiting
   1: GSV(Module,S2,EntryStatus,Local_Slot[2].EntrySts)MEQ(Local_Slot[2].EntrySts,28672,16384)OTE(Local_Slot[2].Running);
   2: [XIO(Local_Slot[2].Running) ,XIC(Local_ModFlts.2) XIO(Sy_ClrFlt) ]OTE(Local_ModFlts.2);
   // ----------AMCI-1242 Module Status ----------
   // Only bits 12-15 are valid.
   // 16#0000 - Standby
   // 16#1000 - Faulted
   // 16#2000 - Validating
   // 16#3000 - Connecting
   // 16#4000 - Running
   // 16#5000 - Shutting Down
   // 16#6000 - Inhibited
   // 16#7000 - Waiting
   3: GSV(Module,S3,EntryStatus,Local_Slot[3].EntrySts)MEQ(Local_Slot[3].EntrySts,28672,16384)OTE(Local_Slot[3].Running);
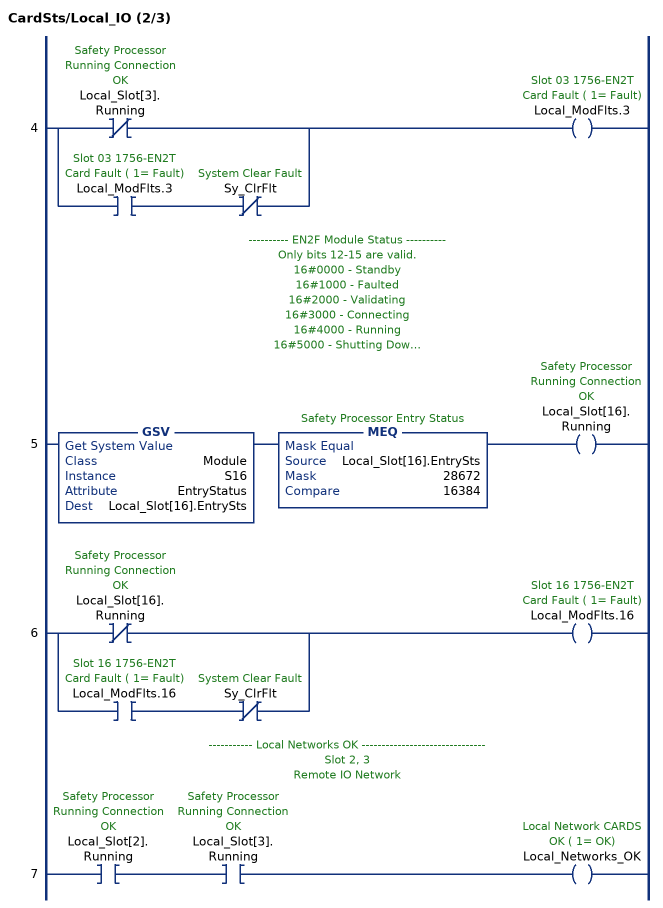
   4: [XIO(Local_Slot[3].Running) ,XIC(Local_ModFlts.3) XIO(Sy_ClrFlt) ]OTE(Local_ModFlts.3);
   // ---------- EN2F Module Status ----------
   // Only bits 12-15 are valid.
   // 16#0000 - Standby
   // 16#1000 - Faulted
   // 16#2000 - Validating
   // 16#3000 - Connecting
   // 16#4000 - Running
   // 16#5000 - Shutting Down
   // 16#6000 - Inhibited
   // 16#7000 - Waiting
   5: GSV(Module,S16,EntryStatus,Local_Slot[16].EntrySts)MEQ(Local_Slot[16].EntrySts,28672,16384)OTE(Local_Slot[16].Running);
   6: [XIO(Local_Slot[16].Running) ,XIC(Local_ModFlts.16) XIO(Sy_ClrFlt) ]OTE(Local_ModFlts.16);
   // ----------- Local Networks OK -------------------------------
   // Slot 2, 3
   // Remote IO Network
   7: XIC(Local_Slot[2].Running)XIC(Local_Slot[3].Running)OTE(Local_Networks_OK);
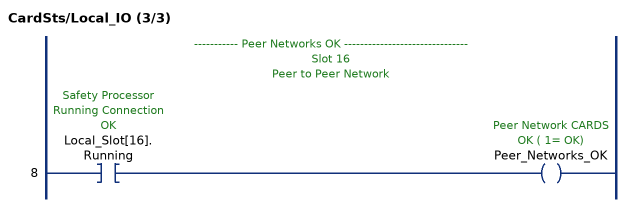
   // ----------- Peer Networks OK -------------------------------
   // Slot 16
   // Peer to Peer Network
   8: XIC(Local_Slot[16].Running)OTE(Peer_Networks_OK);
END_ROUTINE

ROUTINE Main   (* ladder *)
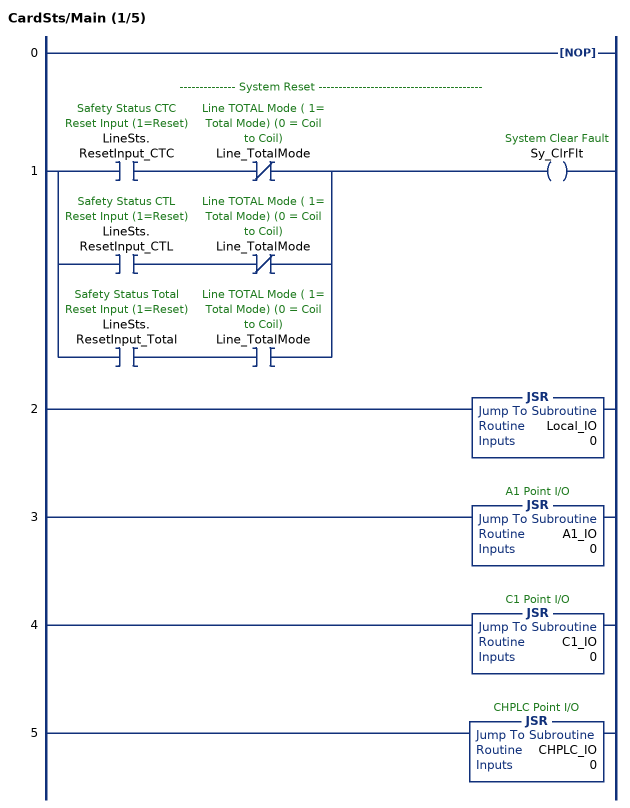
   0: NOP();
   // -------------- System Reset -----------------------------------------
   1: [XIC(LineSts.ResetInput_CTC) XIO(Line_TotalMode) ,XIC(LineSts.ResetInput_CTL) XIO(Line_TotalMode) ,XIC(LineSts.ResetInput_Total) XIC(Line_TotalMode) ]OTE(Sy_ClrFlt);
   2: JSR(Local_IO,0);
   3: JSR(A1_IO,0);
   4: JSR(C1_IO,0);
   5: JSR(CHPLC_IO,0);
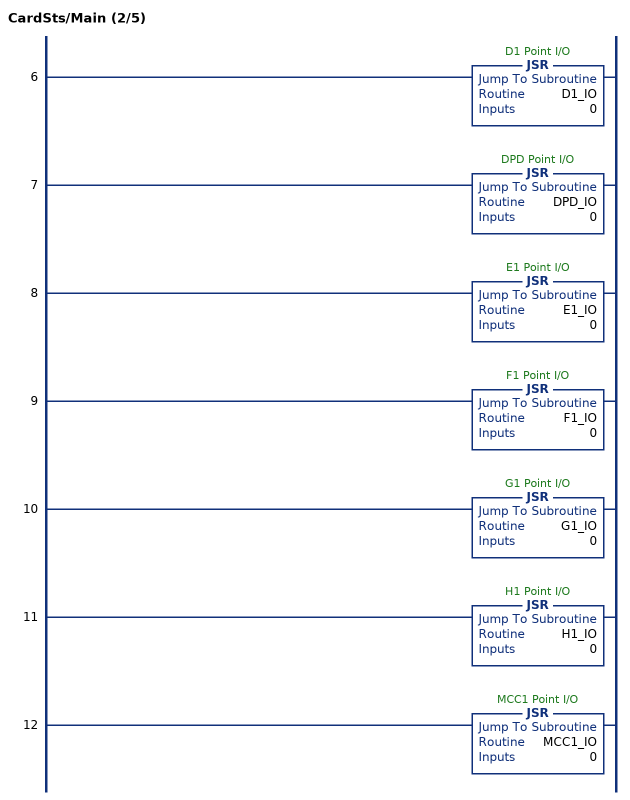
   6: JSR(D1_IO,0);
   7: JSR(DPD_IO,0);
   8: JSR(E1_IO,0);
   9: JSR(F1_IO,0);
   10: JSR(G1_IO,0);
   11: JSR(H1_IO,0);
   12: JSR(MCC1_IO,0);
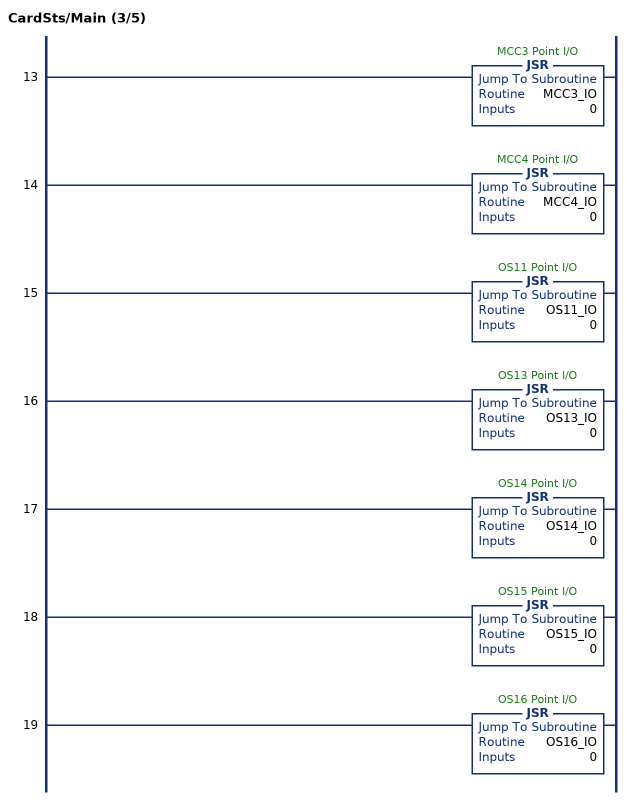
   13: JSR(MCC3_IO,0);
   14: JSR(MCC4_IO,0);
   15: JSR(OS11_IO,0);
   16: JSR(OS13_IO,0);
   17: JSR(OS14_IO,0);
   18: JSR(OS15_IO,0);
   19: JSR(OS16_IO,0);
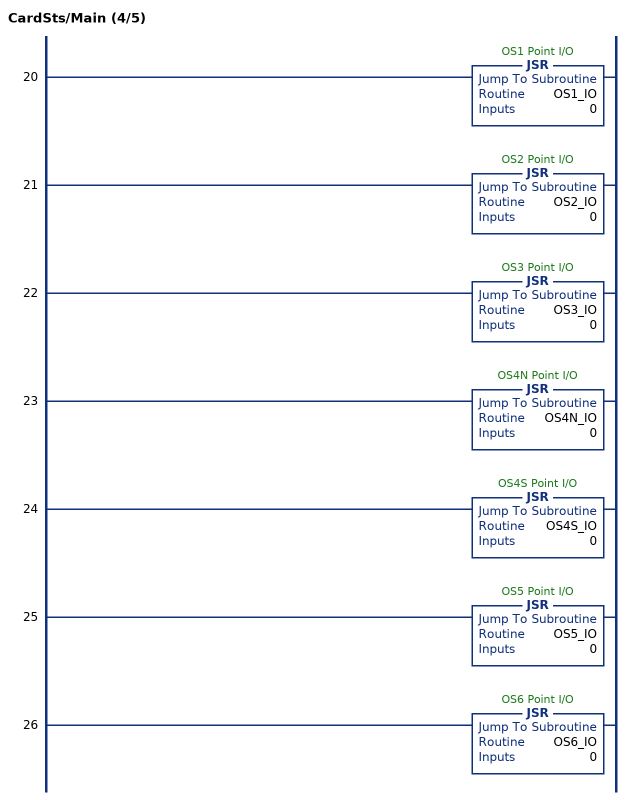
   20: JSR(OS1_IO,0);
   21: JSR(OS2_IO,0);
   22: JSR(OS3_IO,0);
   23: JSR(OS4N_IO,0);
   24: JSR(OS4S_IO,0);
   25: JSR(OS5_IO,0);
   26: JSR(OS6_IO,0);
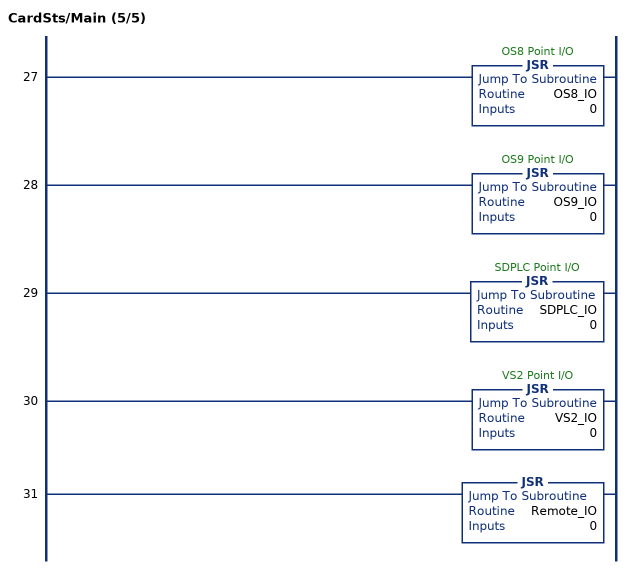
   27: JSR(OS8_IO,0);
   28: JSR(OS9_IO,0);
   29: JSR(SDPLC_IO,0);
   30: JSR(VS2_IO,0);
   31: JSR(Remote_IO,0);
END_ROUTINE

ROUTINE MCC1_IO   (* ladder *)
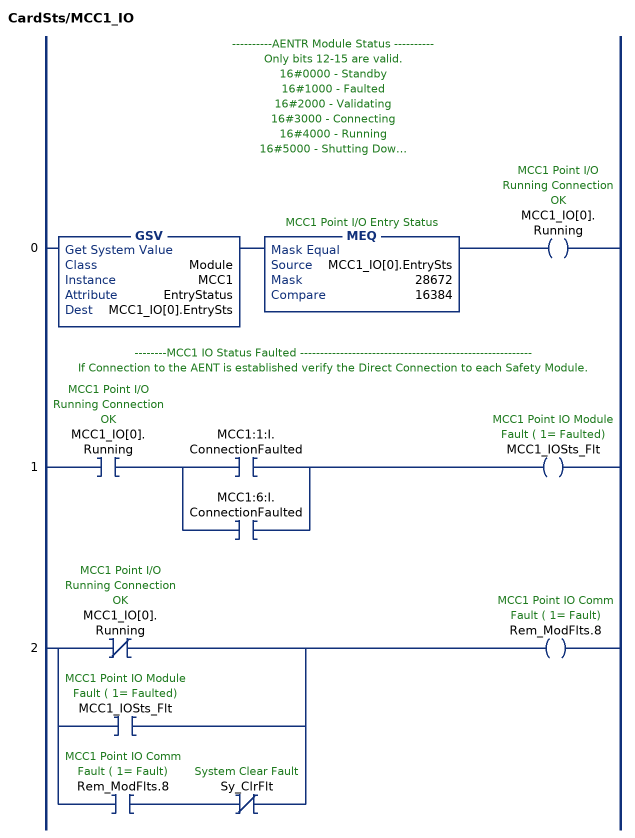
   // ----------AENTR Module Status ----------
   // Only bits 12-15 are valid.
   // 16#0000 - Standby
   // 16#1000 - Faulted
   // 16#2000 - Validating
   // 16#3000 - Connecting
   // 16#4000 - Running
   // 16#5000 - Shutting Down
   // 16#6000 - Inhibited
   // 16#7000 - Waiting
   0: GSV(Module,MCC1,EntryStatus,MCC1_IO[0].EntrySts)MEQ(MCC1_IO[0].EntrySts,28672,16384)OTE(MCC1_IO[0].Running);
   // --------MCC1 IO Status Faulted ----------------------------------------------------------
   // If Connection to the AENT is established verify the Direct Connection to each Safety Module.
   1: XIC(MCC1_IO[0].Running)[XIC(MCC1:1:I.ConnectionFaulted) ,XIC(MCC1:6:I.ConnectionFaulted) ]OTE(MCC1_IOSts_Flt);
   2: [XIO(MCC1_IO[0].Running) ,XIC(MCC1_IOSts_Flt) ,XIC(Rem_ModFlts.8) XIO(Sy_ClrFlt) ]OTE(Rem_ModFlts.8);
END_ROUTINE
